(* Logix 5000 project; controller cal1632 1756-L62 rev 16.20; software revision 16.05; part 20 of 57 *)
(* tags used below, declared in another part *)
   FAULT : BOOL;
   HMI : BOOL;
   p01_param_oven_timer_presets : DINT[32];
   p01_param_process_air_hl : REAL;
   p01_sys_lc : Limit_Clamp;
   p01r09_pb_global_reset : BOOL;
   p02_real_from_hmi : hmi_real;
   p12r31_timer_warning : TIMER[5];
   p12r32_timer_warning : TIMER[5];
   p13_dint_to_hmi : DINT[16];
   p13_param_fast_to_soak : REAL;
   p13_param_lfl_hhl : REAL;
   p13_param_lfl_hl : REAL;
   p13_param_pid1_ff : REAL;
   p13_param_pid1_kd : REAL;
   p13_param_pid1_ki : REAL;
   p13_param_pid1_kp : REAL;
   p13_param_pid2_ff : REAL;
   p13_param_pid2_kd : REAL;
   p13_param_pid2_ki : REAL;
   p13_param_pid2_kp : REAL;
   p13_param_shutdown_temp : REAL;
   p13_param_soak_to_fast : REAL;
   p13_param_tc01_dev : REAL;
   p13_param_tc01_hl : REAL;
   p13_param_tc01z : REAL;
   p13_param_tc02z : REAL;
   p13_param_zone_pressure : REAL;
   p13r02_timer_safe_temp : TIMER[2];
   p13r02_timer_warning : TIMER[4];
   p13r07 : routine;
   p13r07_timer_fault : TIMER[4];
   p13r07_timer_warning : TIMER[4];
   p13r08 : routine;
   p13r08_timer_fault : TIMER[4];
   p13r08_timer_warning : TIMER[4];
   p13r09 : routine;
   p13r09_timer_fault : TIMER[4];
   p13r09_timer_warning : TIMER[8];
   p13r10 : routine;
   p13r10_timer_fault : TIMER[4];
   p13r10_timer_warning : TIMER[4];
   p13r20 : routine;
   p13r20_timer_state_11 : TIMER;
   p13r20_timer_state_3 : TIMER;
   p13r20_timer_state_4 : TIMER;
   p13r20_timer_state_7 : TIMER;
   p13r30 : routine;
   p13r30_cv_man_sp : REAL;
   p13r30_temp_deviation_setpoint : DINT;
   p13r30_timer_fault : TIMER[16];
   p13r30_timer_warning : TIMER[12];
   p13r31 : routine;
   p13r31_timer_fault : TIMER[5];
   p13r31_timer_warning : TIMER[5];
   p13r32 : routine;
   p13r32_timer_fault : TIMER[5];
   p13r32_timer_warning : TIMER[5];
(* P13_Zone_3, continued *)

ROUTINE R07_Alarms   (* ladder *)
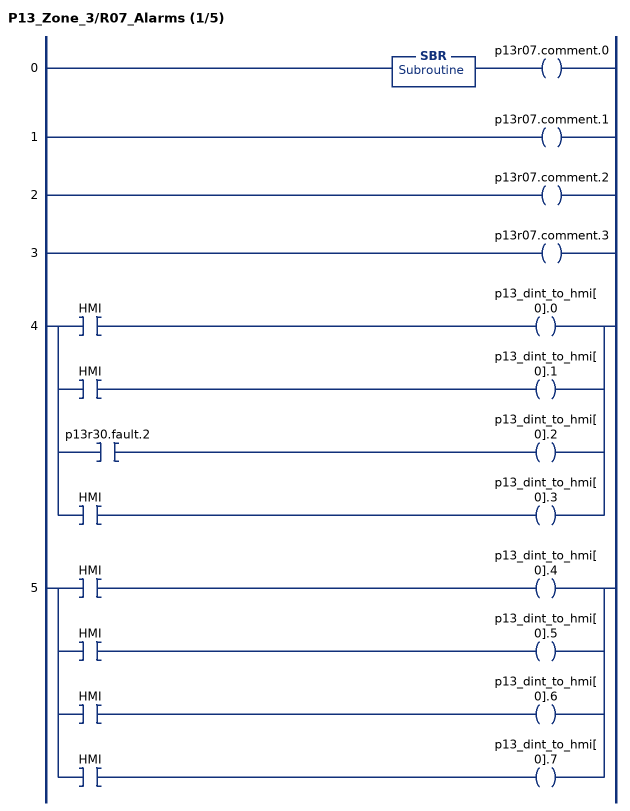
   0: SBR()OTE(p13r07.comment.0);
   1: OTE(p13r07.comment.1);
   2: OTE(p13r07.comment.2);
   3: OTE(p13r07.comment.3);
   4: [XIC(HMI) OTE(p13_dint_to_hmi[0].0) ,XIC(HMI) OTE(p13_dint_to_hmi[0].1) ,XIC(p13r30.fault.2) OTE(p13_dint_to_hmi[0].2) ,XIC(HMI) OTE(p13_dint_to_hmi[0].3) ];
   5: [XIC(HMI) OTE(p13_dint_to_hmi[0].4) ,XIC(HMI) OTE(p13_dint_to_hmi[0].5) ,XIC(HMI) OTE(p13_dint_to_hmi[0].6) ,XIC(HMI) OTE(p13_dint_to_hmi[0].7) ];
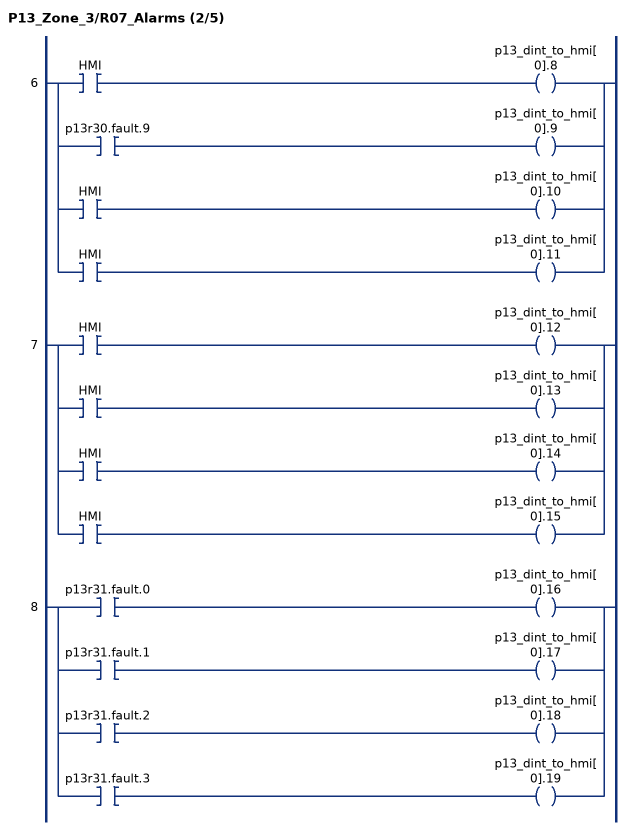
   6: [XIC(HMI) OTE(p13_dint_to_hmi[0].8) ,XIC(p13r30.fault.9) OTE(p13_dint_to_hmi[0].9) ,XIC(HMI) OTE(p13_dint_to_hmi[0].10) ,XIC(HMI) OTE(p13_dint_to_hmi[0].11) ];
   7: [XIC(HMI) OTE(p13_dint_to_hmi[0].12) ,XIC(HMI) OTE(p13_dint_to_hmi[0].13) ,XIC(HMI) OTE(p13_dint_to_hmi[0].14) ,XIC(HMI) OTE(p13_dint_to_hmi[0].15) ];
   8: [XIC(p13r31.fault.0) OTE(p13_dint_to_hmi[0].16) ,XIC(p13r31.fault.1) OTE(p13_dint_to_hmi[0].17) ,XIC(p13r31.fault.2) OTE(p13_dint_to_hmi[0].18) ,XIC(p13r31.fault.3) OTE(p13_dint_to_hmi[0].19) ];
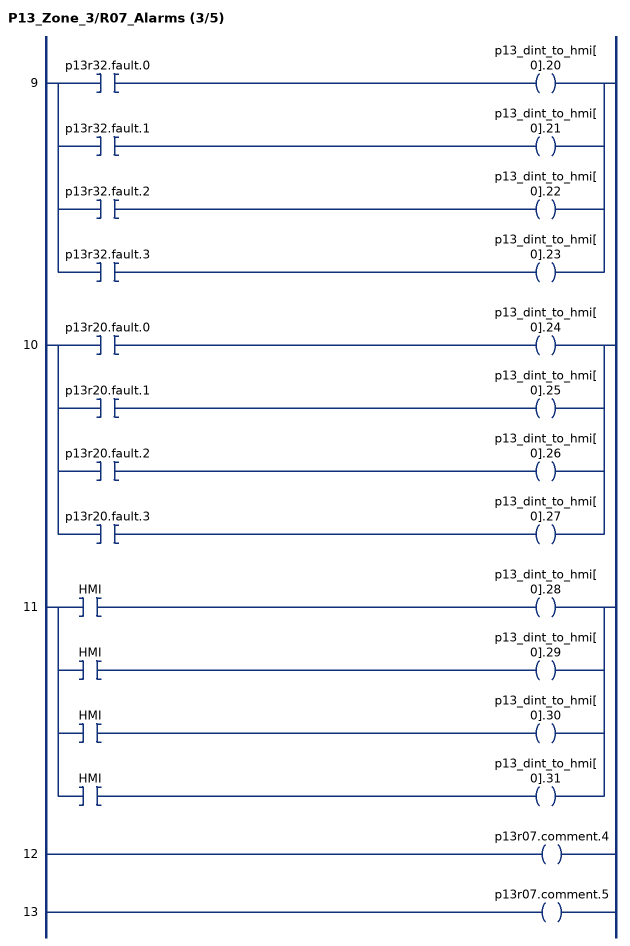
   9: [XIC(p13r32.fault.0) OTE(p13_dint_to_hmi[0].20) ,XIC(p13r32.fault.1) OTE(p13_dint_to_hmi[0].21) ,XIC(p13r32.fault.2) OTE(p13_dint_to_hmi[0].22) ,XIC(p13r32.fault.3) OTE(p13_dint_to_hmi[0].23) ];
   10: [XIC(p13r20.fault.0) OTE(p13_dint_to_hmi[0].24) ,XIC(p13r20.fault.1) OTE(p13_dint_to_hmi[0].25) ,XIC(p13r20.fault.2) OTE(p13_dint_to_hmi[0].26) ,XIC(p13r20.fault.3) OTE(p13_dint_to_hmi[0].27) ];
   11: [XIC(HMI) OTE(p13_dint_to_hmi[0].28) ,XIC(HMI) OTE(p13_dint_to_hmi[0].29) ,XIC(HMI) OTE(p13_dint_to_hmi[0].30) ,XIC(HMI) OTE(p13_dint_to_hmi[0].31) ];
   12: OTE(p13r07.comment.4);
   13: OTE(p13r07.comment.5);
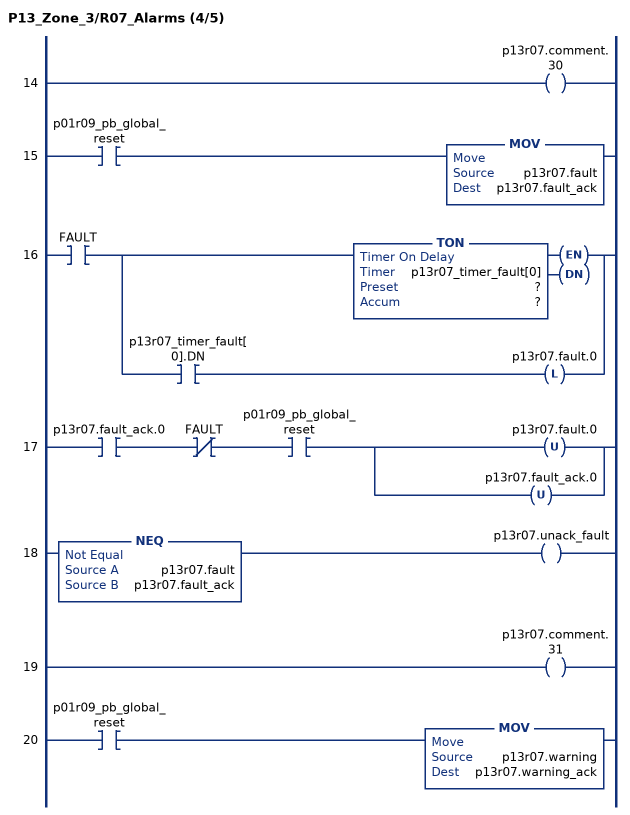
   14: OTE(p13r07.comment.30);
   15: XIC(p01r09_pb_global_reset)MOV(p13r07.fault,p13r07.fault_ack);
   16: XIC(FAULT)[TON(p13r07_timer_fault[0],?,?) ,XIC(p13r07_timer_fault[0].DN) OTL(p13r07.fault.0) ];
   17: XIC(p13r07.fault_ack.0)XIO(FAULT)XIC(p01r09_pb_global_reset)[OTU(p13r07.fault.0) ,OTU(p13r07.fault_ack.0) ];
   18: NEQ(p13r07.fault,p13r07.fault_ack)OTE(p13r07.unack_fault);
   19: OTE(p13r07.comment.31);
   20: XIC(p01r09_pb_global_reset)MOV(p13r07.warning,p13r07.warning_ack);
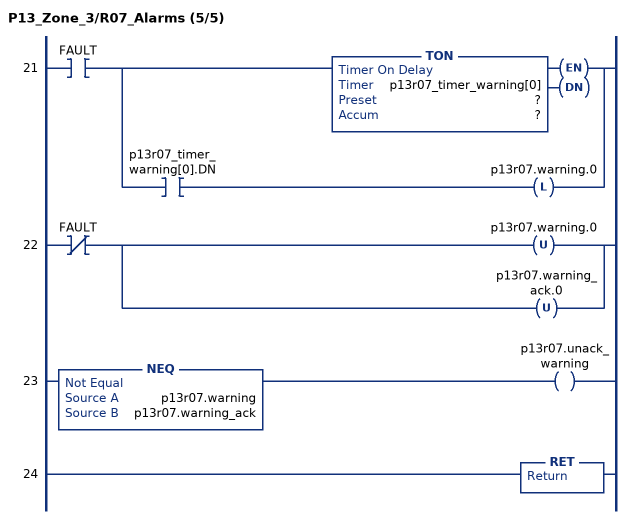
   21: XIC(FAULT)[TON(p13r07_timer_warning[0],?,?) ,XIC(p13r07_timer_warning[0].DN) OTL(p13r07.warning.0) ];
   22: XIO(FAULT)[OTU(p13r07.warning.0) ,OTU(p13r07.warning_ack.0) ];
   23: NEQ(p13r07.warning,p13r07.warning_ack)OTE(p13r07.unack_warning);
   24: RET();
END_ROUTINE

ROUTINE R08_Warnings   (* ladder *)
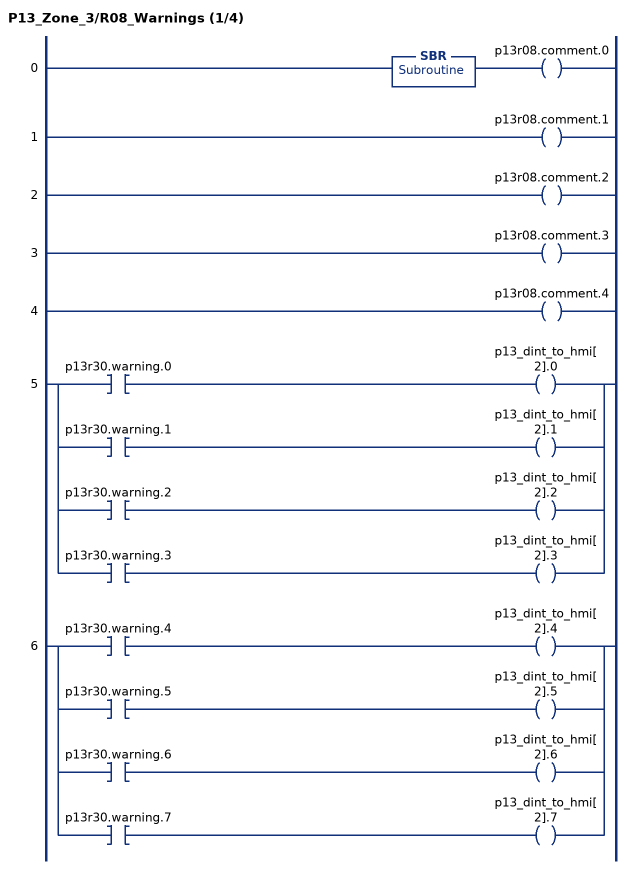
   0: SBR()OTE(p13r08.comment.0);
   1: OTE(p13r08.comment.1);
   2: OTE(p13r08.comment.2);
   3: OTE(p13r08.comment.3);
   4: OTE(p13r08.comment.4);
   5: [XIC(p13r30.warning.0) OTE(p13_dint_to_hmi[2].0) ,XIC(p13r30.warning.1) OTE(p13_dint_to_hmi[2].1) ,XIC(p13r30.warning.2) OTE(p13_dint_to_hmi[2].2) ,XIC(p13r30.warning.3) OTE(p13_dint_to_hmi[2].3) ];
   6: [XIC(p13r30.warning.4) OTE(p13_dint_to_hmi[2].4) ,XIC(p13r30.warning.5) OTE(p13_dint_to_hmi[2].5) ,XIC(p13r30.warning.6) OTE(p13_dint_to_hmi[2].6) ,XIC(p13r30.warning.7) OTE(p13_dint_to_hmi[2].7) ];
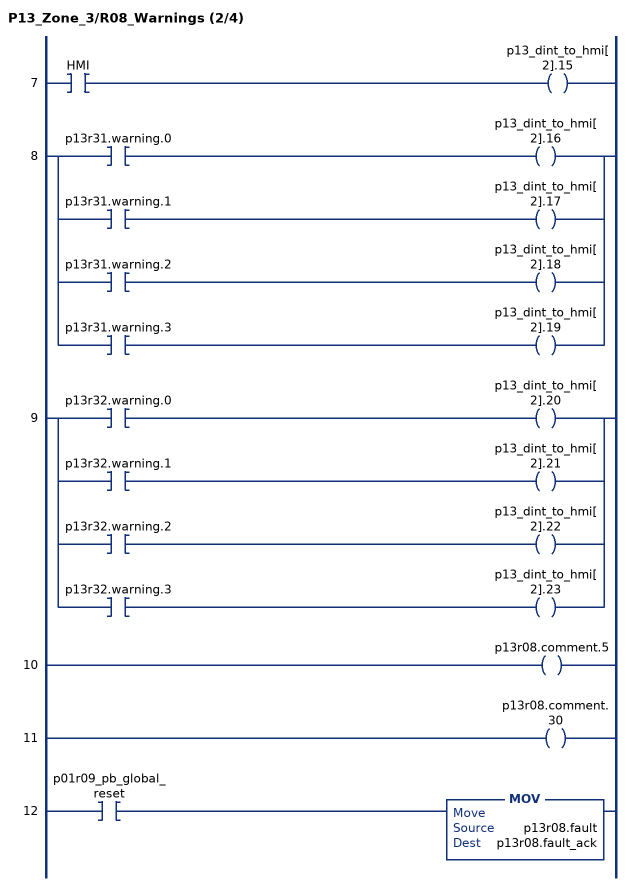
   7: XIC(HMI)OTE(p13_dint_to_hmi[2].15);
   8: [XIC(p13r31.warning.0) OTE(p13_dint_to_hmi[2].16) ,XIC(p13r31.warning.1) OTE(p13_dint_to_hmi[2].17) ,XIC(p13r31.warning.2) OTE(p13_dint_to_hmi[2].18) ,XIC(p13r31.warning.3) OTE(p13_dint_to_hmi[2].19) ];
   9: [XIC(p13r32.warning.0) OTE(p13_dint_to_hmi[2].20) ,XIC(p13r32.warning.1) OTE(p13_dint_to_hmi[2].21) ,XIC(p13r32.warning.2) OTE(p13_dint_to_hmi[2].22) ,XIC(p13r32.warning.3) OTE(p13_dint_to_hmi[2].23) ];
   10: OTE(p13r08.comment.5);
   11: OTE(p13r08.comment.30);
   12: XIC(p01r09_pb_global_reset)MOV(p13r08.fault,p13r08.fault_ack);
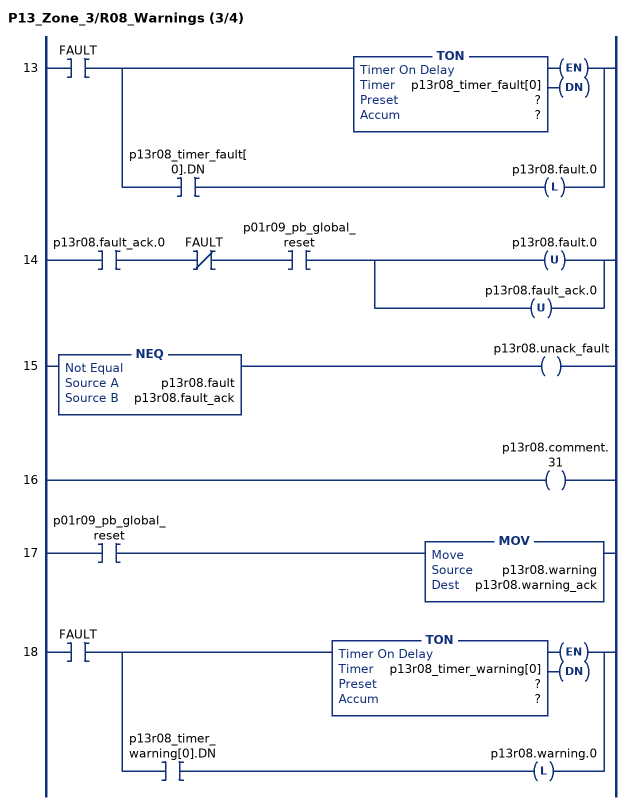
   13: XIC(FAULT)[TON(p13r08_timer_fault[0],?,?) ,XIC(p13r08_timer_fault[0].DN) OTL(p13r08.fault.0) ];
   14: XIC(p13r08.fault_ack.0)XIO(FAULT)XIC(p01r09_pb_global_reset)[OTU(p13r08.fault.0) ,OTU(p13r08.fault_ack.0) ];
   15: NEQ(p13r08.fault,p13r08.fault_ack)OTE(p13r08.unack_fault);
   16: OTE(p13r08.comment.31);
   17: XIC(p01r09_pb_global_reset)MOV(p13r08.warning,p13r08.warning_ack);
   18: XIC(FAULT)[TON(p13r08_timer_warning[0],?,?) ,XIC(p13r08_timer_warning[0].DN) OTL(p13r08.warning.0) ];
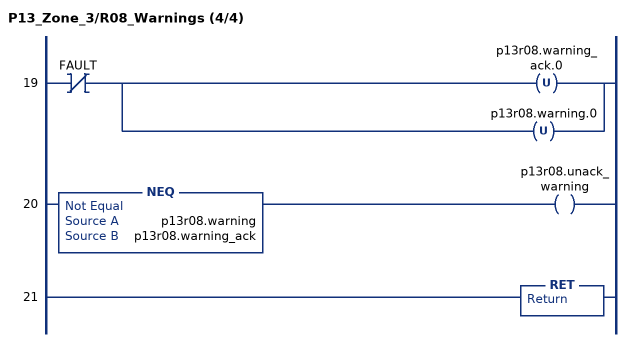
   19: XIO(FAULT)[OTU(p13r08.warning_ack.0) ,OTU(p13r08.warning.0) ];
   20: NEQ(p13r08.warning,p13r08.warning_ack)OTE(p13r08.unack_warning);
   21: RET();
END_ROUTINE

ROUTINE R09_Modes   (* ladder *)
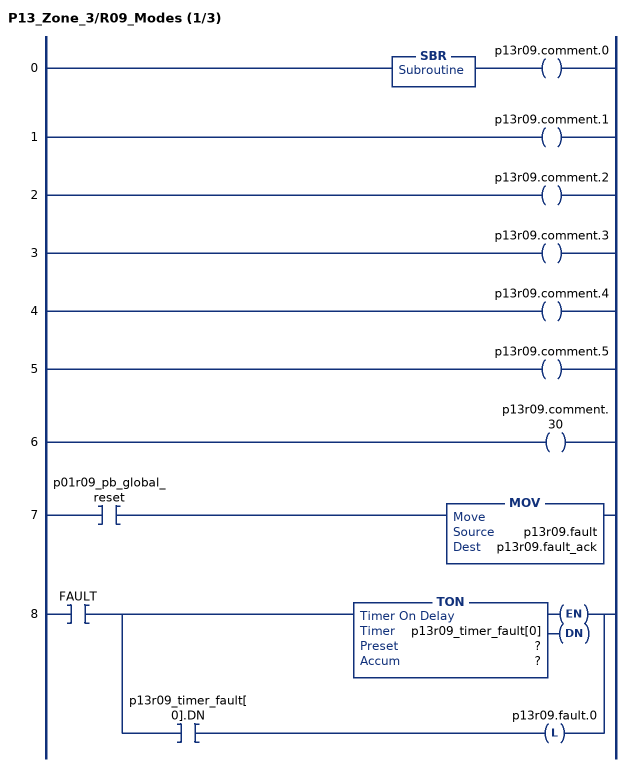
   0: SBR()OTE(p13r09.comment.0);
   1: OTE(p13r09.comment.1);
   2: OTE(p13r09.comment.2);
   3: OTE(p13r09.comment.3);
   4: OTE(p13r09.comment.4);
   5: OTE(p13r09.comment.5);
   6: OTE(p13r09.comment.30);
   7: XIC(p01r09_pb_global_reset)MOV(p13r09.fault,p13r09.fault_ack);
   8: XIC(FAULT)[TON(p13r09_timer_fault[0],?,?) ,XIC(p13r09_timer_fault[0].DN) OTL(p13r09.fault.0) ];
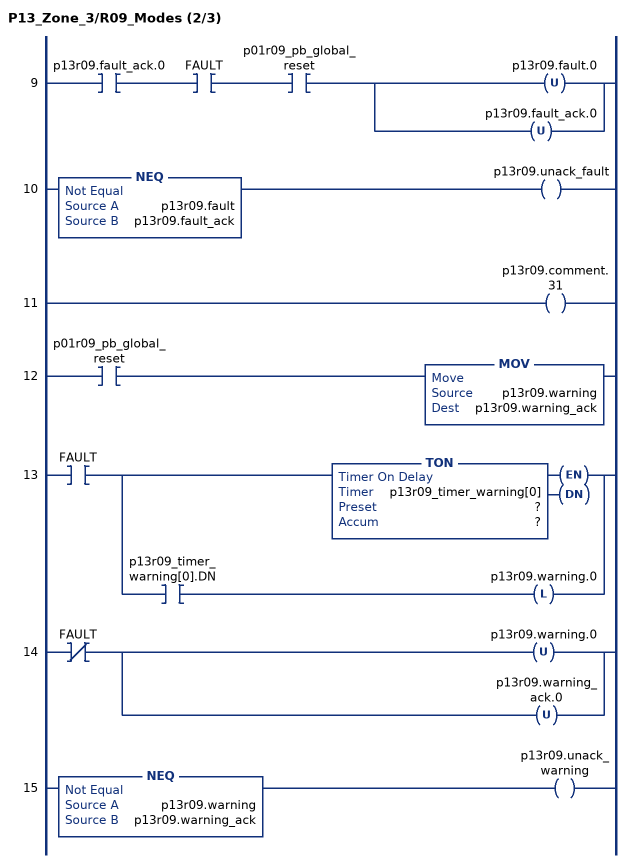
   9: XIC(p13r09.fault_ack.0)XIC(FAULT)XIC(p01r09_pb_global_reset)[OTU(p13r09.fault.0) ,OTU(p13r09.fault_ack.0) ];
   10: NEQ(p13r09.fault,p13r09.fault_ack)OTE(p13r09.unack_fault);
   11: OTE(p13r09.comment.31);
   12: XIC(p01r09_pb_global_reset)MOV(p13r09.warning,p13r09.warning_ack);
   13: XIC(FAULT)[TON(p13r09_timer_warning[0],?,?) ,XIC(p13r09_timer_warning[0].DN) OTL(p13r09.warning.0) ];
   14: XIO(FAULT)[OTU(p13r09.warning.0) ,OTU(p13r09.warning_ack.0) ];
   15: NEQ(p13r09.warning,p13r09.warning_ack)OTE(p13r09.unack_warning);
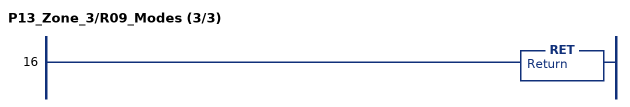
   16: RET();
END_ROUTINE

ROUTINE R10_Parameters   (* ladder *)
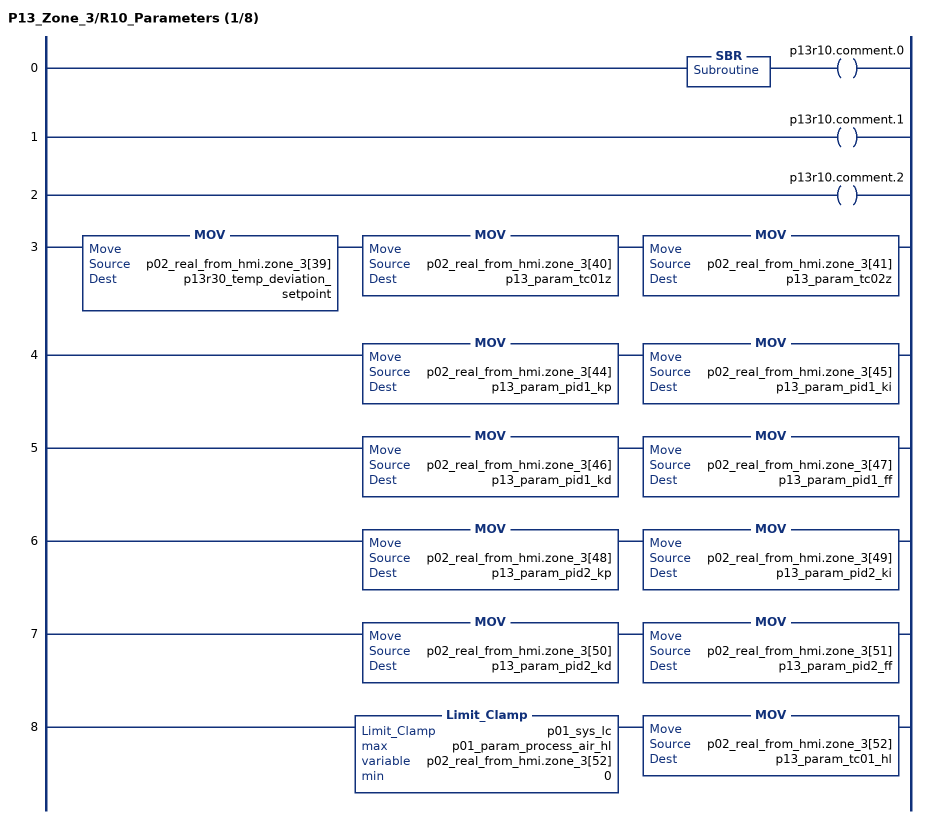
   0: SBR()OTE(p13r10.comment.0);
   1: OTE(p13r10.comment.1);
   2: OTE(p13r10.comment.2);
   3: MOV(p02_real_from_hmi.zone_3[39],p13r30_temp_deviation_setpoint)MOV(p02_real_from_hmi.zone_3[40],p13_param_tc01z)MOV(p02_real_from_hmi.zone_3[41],p13_param_tc02z);
   4: MOV(p02_real_from_hmi.zone_3[44],p13_param_pid1_kp)MOV(p02_real_from_hmi.zone_3[45],p13_param_pid1_ki);
   5: MOV(p02_real_from_hmi.zone_3[46],p13_param_pid1_kd)MOV(p02_real_from_hmi.zone_3[47],p13_param_pid1_ff);
   6: MOV(p02_real_from_hmi.zone_3[48],p13_param_pid2_kp)MOV(p02_real_from_hmi.zone_3[49],p13_param_pid2_ki);
   7: MOV(p02_real_from_hmi.zone_3[50],p13_param_pid2_kd)MOV(p02_real_from_hmi.zone_3[51],p13_param_pid2_ff);
   8: Limit_Clamp(p01_sys_lc,p01_param_process_air_hl,p02_real_from_hmi.zone_3[52],0)MOV(p02_real_from_hmi.zone_3[52],p13_param_tc01_hl);
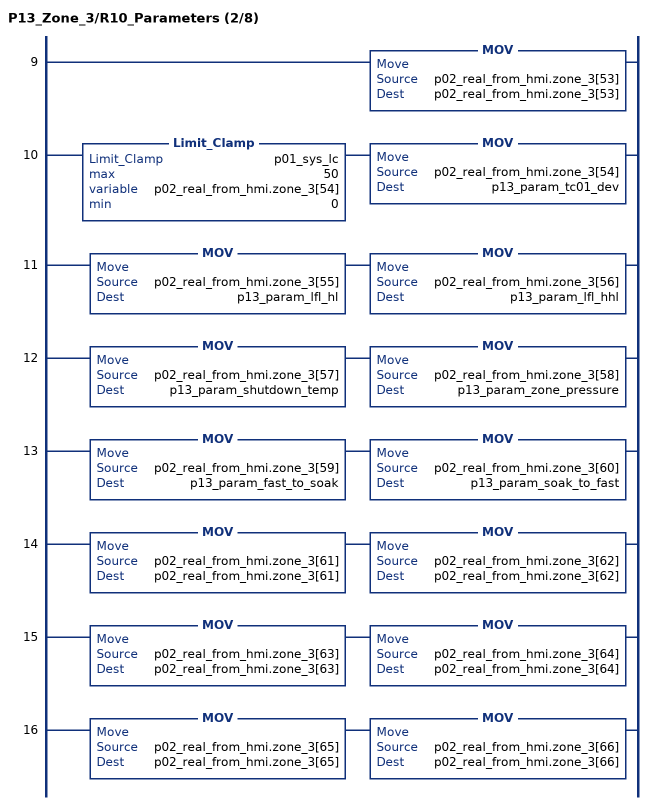
   9: MOV(p02_real_from_hmi.zone_3[53],p02_real_from_hmi.zone_3[53]);
   10: Limit_Clamp(p01_sys_lc,50,p02_real_from_hmi.zone_3[54],0)MOV(p02_real_from_hmi.zone_3[54],p13_param_tc01_dev);
   11: MOV(p02_real_from_hmi.zone_3[55],p13_param_lfl_hl)MOV(p02_real_from_hmi.zone_3[56],p13_param_lfl_hhl);
   12: MOV(p02_real_from_hmi.zone_3[57],p13_param_shutdown_temp)MOV(p02_real_from_hmi.zone_3[58],p13_param_zone_pressure);
   13: MOV(p02_real_from_hmi.zone_3[59],p13_param_fast_to_soak)MOV(p02_real_from_hmi.zone_3[60],p13_param_soak_to_fast);
   14: MOV(p02_real_from_hmi.zone_3[61],p02_real_from_hmi.zone_3[61])MOV(p02_real_from_hmi.zone_3[62],p02_real_from_hmi.zone_3[62]);
   15: MOV(p02_real_from_hmi.zone_3[63],p02_real_from_hmi.zone_3[63])MOV(p02_real_from_hmi.zone_3[64],p02_real_from_hmi.zone_3[64]);
   16: MOV(p02_real_from_hmi.zone_3[65],p02_real_from_hmi.zone_3[65])MOV(p02_real_from_hmi.zone_3[66],p02_real_from_hmi.zone_3[66]);
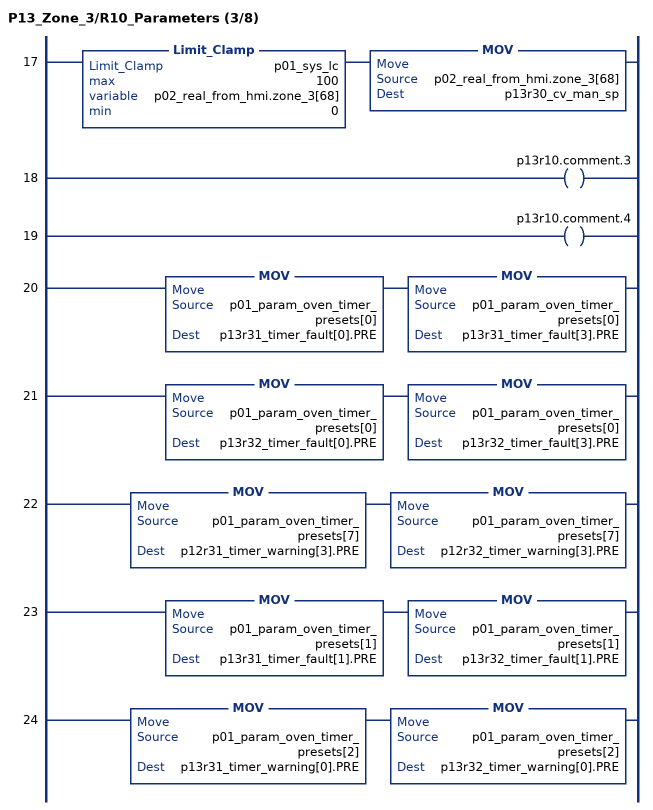
   17: Limit_Clamp(p01_sys_lc,100,p02_real_from_hmi.zone_3[68],0)MOV(p02_real_from_hmi.zone_3[68],p13r30_cv_man_sp);
   18: OTE(p13r10.comment.3);
   19: OTE(p13r10.comment.4);
   20: MOV(p01_param_oven_timer_presets[0],p13r31_timer_fault[0].PRE)MOV(p01_param_oven_timer_presets[0],p13r31_timer_fault[3].PRE);
   21: MOV(p01_param_oven_timer_presets[0],p13r32_timer_fault[0].PRE)MOV(p01_param_oven_timer_presets[0],p13r32_timer_fault[3].PRE);
   22: MOV(p01_param_oven_timer_presets[7],p12r31_timer_warning[3].PRE)MOV(p01_param_oven_timer_presets[7],p12r32_timer_warning[3].PRE);
   23: MOV(p01_param_oven_timer_presets[1],p13r31_timer_fault[1].PRE)MOV(p01_param_oven_timer_presets[1],p13r32_timer_fault[1].PRE);
   24: MOV(p01_param_oven_timer_presets[2],p13r31_timer_warning[0].PRE)MOV(p01_param_oven_timer_presets[2],p13r32_timer_warning[0].PRE);
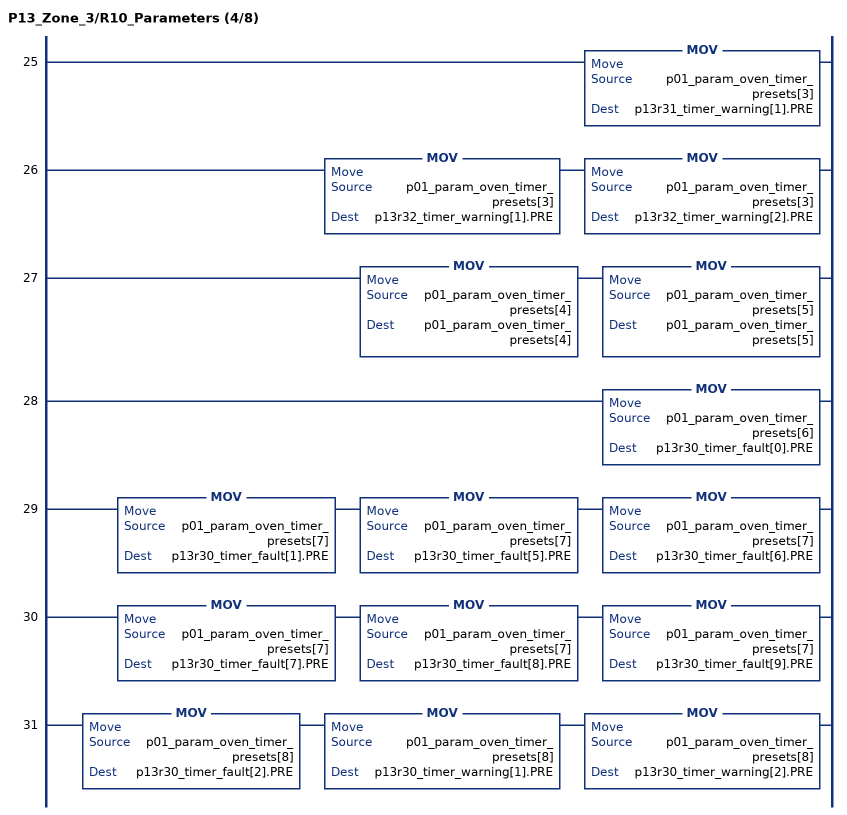
   25: MOV(p01_param_oven_timer_presets[3],p13r31_timer_warning[1].PRE);
   26: MOV(p01_param_oven_timer_presets[3],p13r32_timer_warning[1].PRE)MOV(p01_param_oven_timer_presets[3],p13r32_timer_warning[2].PRE);
   27: MOV(p01_param_oven_timer_presets[4],p01_param_oven_timer_presets[4])MOV(p01_param_oven_timer_presets[5],p01_param_oven_timer_presets[5]);
   28: MOV(p01_param_oven_timer_presets[6],p13r30_timer_fault[0].PRE);
   29: MOV(p01_param_oven_timer_presets[7],p13r30_timer_fault[1].PRE)MOV(p01_param_oven_timer_presets[7],p13r30_timer_fault[5].PRE)MOV(p01_param_oven_timer_presets[7],p13r30_timer_fault[6].PRE);
   30: MOV(p01_param_oven_timer_presets[7],p13r30_timer_fault[7].PRE)MOV(p01_param_oven_timer_presets[7],p13r30_timer_fault[8].PRE)MOV(p01_param_oven_timer_presets[7],p13r30_timer_fault[9].PRE);
   31: MOV(p01_param_oven_timer_presets[8],p13r30_timer_fault[2].PRE)MOV(p01_param_oven_timer_presets[8],p13r30_timer_warning[1].PRE)MOV(p01_param_oven_timer_presets[8],p13r30_timer_warning[2].PRE);
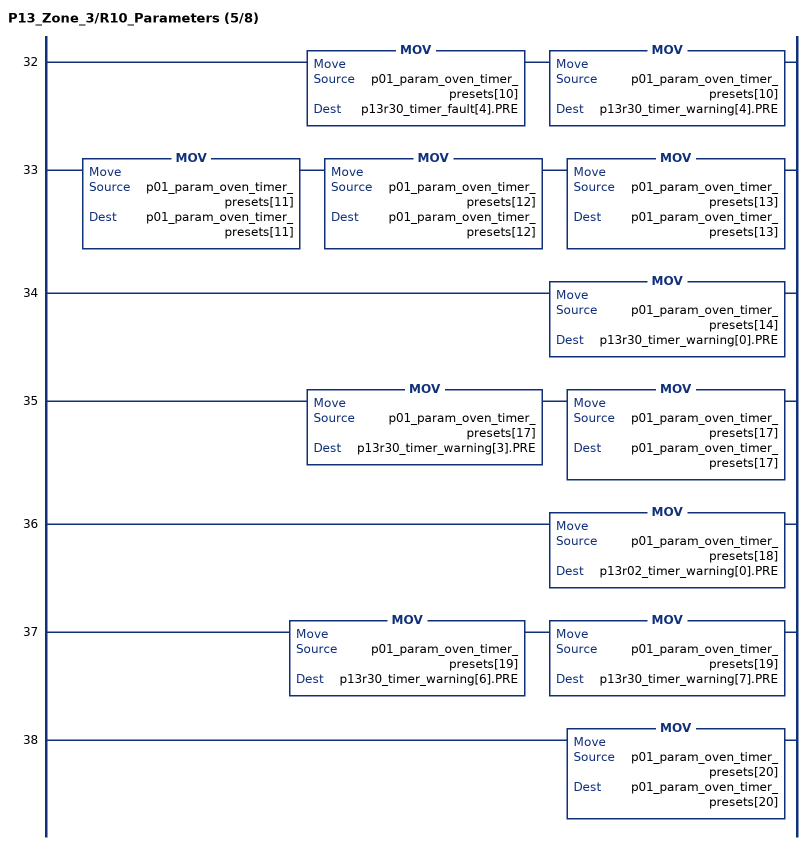
   32: MOV(p01_param_oven_timer_presets[10],p13r30_timer_fault[4].PRE)MOV(p01_param_oven_timer_presets[10],p13r30_timer_warning[4].PRE);
   33: MOV(p01_param_oven_timer_presets[11],p01_param_oven_timer_presets[11])MOV(p01_param_oven_timer_presets[12],p01_param_oven_timer_presets[12])MOV(p01_param_oven_timer_presets[13],p01_param_oven_timer_presets[13]);
   34: MOV(p01_param_oven_timer_presets[14],p13r30_timer_warning[0].PRE);
   35: MOV(p01_param_oven_timer_presets[17],p13r30_timer_warning[3].PRE)MOV(p01_param_oven_timer_presets[17],p01_param_oven_timer_presets[17]);
   36: MOV(p01_param_oven_timer_presets[18],p13r02_timer_warning[0].PRE);
   37: MOV(p01_param_oven_timer_presets[19],p13r30_timer_warning[6].PRE)MOV(p01_param_oven_timer_presets[19],p13r30_timer_warning[7].PRE);
   38: MOV(p01_param_oven_timer_presets[20],p01_param_oven_timer_presets[20]);
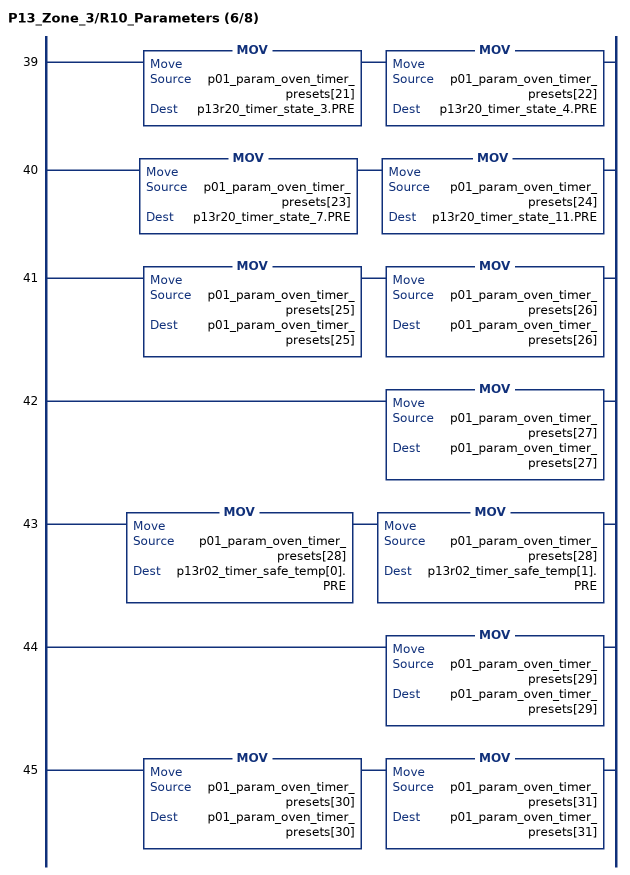
   39: MOV(p01_param_oven_timer_presets[21],p13r20_timer_state_3.PRE)MOV(p01_param_oven_timer_presets[22],p13r20_timer_state_4.PRE);
   40: MOV(p01_param_oven_timer_presets[23],p13r20_timer_state_7.PRE)MOV(p01_param_oven_timer_presets[24],p13r20_timer_state_11.PRE);
   41: MOV(p01_param_oven_timer_presets[25],p01_param_oven_timer_presets[25])MOV(p01_param_oven_timer_presets[26],p01_param_oven_timer_presets[26]);
   42: MOV(p01_param_oven_timer_presets[27],p01_param_oven_timer_presets[27]);
   43: MOV(p01_param_oven_timer_presets[28],p13r02_timer_safe_temp[0].PRE)MOV(p01_param_oven_timer_presets[28],p13r02_timer_safe_temp[1].PRE);
   44: MOV(p01_param_oven_timer_presets[29],p01_param_oven_timer_presets[29]);
   45: MOV(p01_param_oven_timer_presets[30],p01_param_oven_timer_presets[30])MOV(p01_param_oven_timer_presets[31],p01_param_oven_timer_presets[31]);
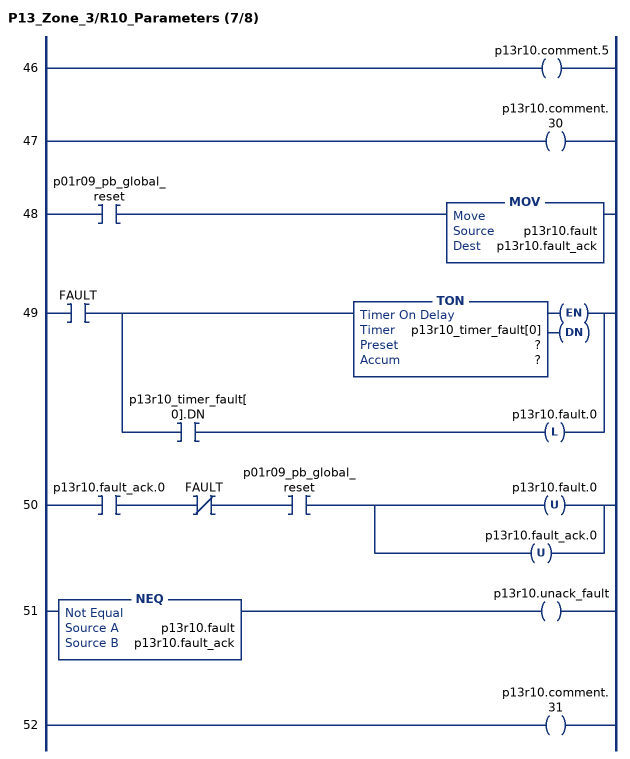
   46: OTE(p13r10.comment.5);
   47: OTE(p13r10.comment.30);
   48: XIC(p01r09_pb_global_reset)MOV(p13r10.fault,p13r10.fault_ack);
   49: XIC(FAULT)[TON(p13r10_timer_fault[0],?,?) ,XIC(p13r10_timer_fault[0].DN) OTL(p13r10.fault.0) ];
   50: XIC(p13r10.fault_ack.0)XIO(FAULT)XIC(p01r09_pb_global_reset)[OTU(p13r10.fault.0) ,OTU(p13r10.fault_ack.0) ];
   51: NEQ(p13r10.fault,p13r10.fault_ack)OTE(p13r10.unack_fault);
   52: OTE(p13r10.comment.31);
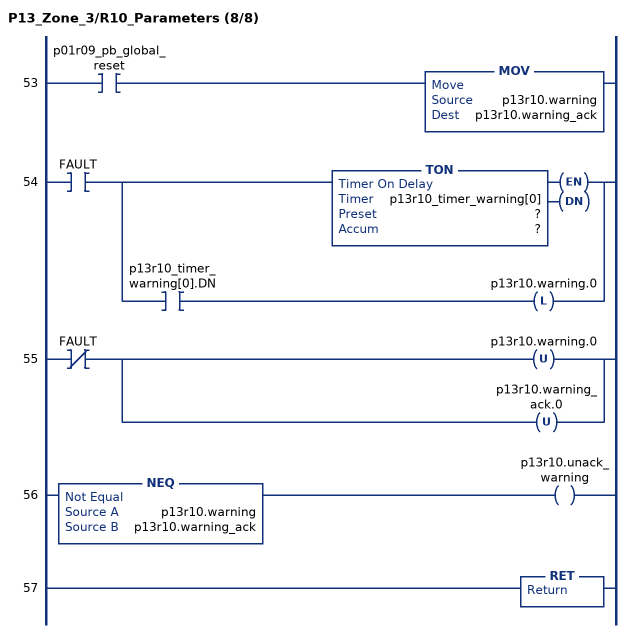
   53: XIC(p01r09_pb_global_reset)MOV(p13r10.warning,p13r10.warning_ack);
   54: XIC(FAULT)[TON(p13r10_timer_warning[0],?,?) ,XIC(p13r10_timer_warning[0].DN) OTL(p13r10.warning.0) ];
   55: XIO(FAULT)[OTU(p13r10.warning.0) ,OTU(p13r10.warning_ack.0) ];
   56: NEQ(p13r10.warning,p13r10.warning_ack)OTE(p13r10.unack_warning);
   57: RET();
END_ROUTINE
